// TIA Portal project "Traffic_feu" (V15)

(* hardware
DEVICE "Station S7-1200_1"  S7-1200 Station
   slot 0: "Châssis_0"  S7-1200 Rack  Rack  V1.0
   slot 1: "PLC_1"  CPU 1215C AC/DC/Rly  6ES7 215-1BG40-0XB0  V4.2
DEVICE "HMI_1"  KTP700 Basic PN
   slot 0: "HMI_1"  KTP700 Basic PN  6AV2 123-2GB03-0AX0  15.0.0.0
   slot 1: "HMI_RT_1"  KTP700 Basic PN  6AV2 123-2GB03-0AX0  15.0.0.0
   slot 5: "HMI_1.IE_CP_1"  PROFINET Interface  15.0.0.0
      slot 1: "Interface PROFINET_1"  PROFINET Interface
         slot 1: "Port_1"  Port
*)

// ===== PLC "PLC_1"  CPU 1215C AC/DC/Rly =====

VAR_GLOBAL   // PLC tag table "Table de variables standard"
   "TAG" AT %Q0.3 : Bool;
END_VAR

VAR_GLOBAL   // PLC tag table "table_feux"
   "Marche" AT %M0.0 : Bool;
   "feu_vert" AT %Q0.0 : Bool;
   "feu_orange" AT %Q0.1 : Bool;
   "feu_rouge" AT %Q0.2 : Bool;
END_VAR

DATA_BLOCK "Bloc_1_DB_1"   // DB5
{ S7_Optimized_Access := 'TRUE' }
VERSION : 0.1
// stored: InstanceOfName Bloc_1
"Bloc_1"
BEGIN
END_DATA_BLOCK

// folder: System blocks/Program resources

DATA_BLOCK "T_vert"   // DB1
{ S7_Optimized_Access := 'TRUE' }
AUTHOR : Simatic
FAMILY : IEC
NAME : IEC_TMR
VERSION : 1.0
// stored: InstanceOfName IEC_TIMER
"IEC_TIMER"
BEGIN
END_DATA_BLOCK

DATA_BLOCK "t_orange"   // DB2
{ S7_Optimized_Access := 'TRUE' }
AUTHOR : Simatic
FAMILY : IEC
NAME : IEC_TMR
VERSION : 1.0
// stored: InstanceOfName IEC_TIMER
"IEC_TIMER"
BEGIN
END_DATA_BLOCK

DATA_BLOCK "t_rouge"   // DB3
{ S7_Optimized_Access := 'TRUE' }
AUTHOR : Simatic
FAMILY : IEC
NAME : IEC_TMR
VERSION : 1.0
// stored: InstanceOfName IEC_TIMER
"IEC_TIMER"
BEGIN
END_DATA_BLOCK

// folder: (top level)

FUNCTION_BLOCK "Bloc_1"   // FB1, LAD
{ S7_Optimized_Access := 'TRUE' }
VERSION : 0.1
BEGIN

REGION Network 1
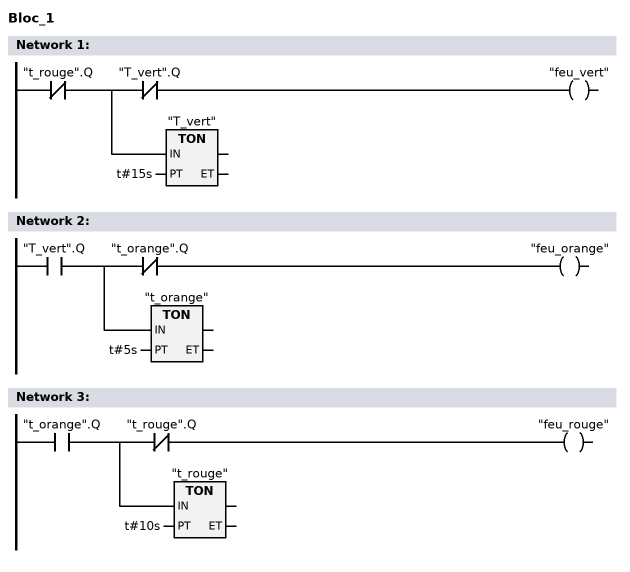
   "feu_vert" := NOT "t_rouge".Q AND NOT "T_vert".Q;
   "T_vert".TON(IN := NOT "t_rouge".Q, PT := t#15s);
END_REGION

REGION Network 2
   "feu_orange" := "T_vert".Q AND NOT "t_orange".Q;
   "t_orange".TON(IN := "T_vert".Q, PT := t#5s);
END_REGION

REGION Network 3
   "feu_rouge" := "t_orange".Q AND NOT "t_rouge".Q;
   "t_rouge".TON(IN := "t_orange".Q, PT := t#10s);
END_REGION
END_FUNCTION_BLOCK

ORGANIZATION_BLOCK "Main"   // OB1, LAD, ProgramCycle
TITLE = "Main Program Sweep (Cycle)"
{ S7_Optimized_Access := 'TRUE' }
VERSION : 0.1
   VAR_INPUT
      Initial_Call : Bool;   // Initial call of this OB
      Remanence : Bool;   // =True, if remanent data are available
   END_VAR
BEGIN

REGION Network 1
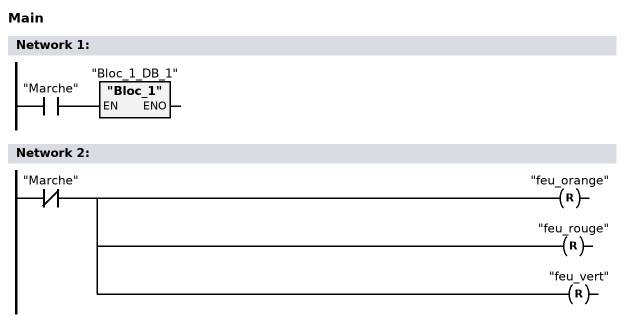
   RUNG wire#powerrail
      Contact( "Marche" )
      "Bloc_1_DB_1"()
   END_RUNG
   // the same network as SCL:
   IF "Marche" THEN
       "Bloc_1_DB_1"();   // "Bloc_1"
   END_IF;
END_REGION

REGION Network 2
   RUNG wire#powerrail
      I_Contact( "Marche" )
      wire#w1
      R_Coil( "feu_orange" )
   END_RUNG
   RUNG wire#w1
      R_Coil( "feu_rouge" )
   END_RUNG
   RUNG wire#w1
      R_Coil( "feu_vert" )
   END_RUNG
   // the same network as SCL:
   IF NOT "Marche" THEN
       "feu_orange" := FALSE;
       "feu_rouge" := FALSE;
       "feu_vert" := FALSE;
   END_IF;
END_REGION
END_ORGANIZATION_BLOCK

(* ===== HMI "HMI_RT_1" =====
system functions are stored by id; their names below are inferred from use
connection "HMI_Liaison_1": ETHERNET, SMART_S7_1200_OMS

HMI tags "Table de variables standard"
   "Numéro_vue_variable" : UInt, internal
   "vert_IHM_1" : Bool = PLC feu_vert AT %Q0.0, 1 s
   "orange_IHM_1" : Bool = PLC feu_orange AT %Q0.1, 1 s
   "rouge_IHM_1" : Bool = PLC feu_rouge AT %Q0.2, 1 s
   "rouge_IHM_1(1)" : Bool = PLC feu_rouge AT %Q0.2, 1 s
   "Marche" : Bool = PLC Marche AT %M0.0, 1 s

text list "Nom_vue_liste_textes": 1 'Vue racine'

Template "Modèle_1" 800x480
   SymbolicIOField "Vue_champ_ES_symbolique" at 2,9 size 691x33; TextOff '0'; TextOn '1'; TextList "Nom_vue_liste_textes"
      ProcessValue <- "Numéro_vue_variable"
      on Change: ActivateScreenByNumber("Numéro_vue_variable", 0)
   DateTimeField "HmiScreenItemData" at 695,25 size 105x25
   DateTimeField "HmiScreenItemData_1" at 695,0 size 105x25

screen "Vue racine" 800x480, template "Modèle_1"
   on GenerateScreen: SetTag("Numéro_vue_variable", 1)
   Circle "Cercle_1" at 312,109 size 57x57
      Appearance <- "vert_IHM_1"
   Circle "Cercle_2" at 311,164 size 57x57
      Appearance <- "orange_IHM_1"
   Circle "Cercle_3" at 311,221 size 57x57
      Appearance <- "rouge_IHM_1(1)"
   Button "Bouton_1" at 60,135 size 105x44; TextOff 'Start'
      on Press: SetBit("Marche")
   Button "Bouton_2" at 60,200 size 105x44; TextOff 'Stop'
      on Press: ResetBit("Marche")
   GraphicView "Vue de graphique_1" at 300,272 size 77x112; Picture "Graphique_1"
*)